FUNCTION_BLOCK FB_VISU_STOP_GATE
VAR_INPUT
END_VAR
VAR_OUTPUT
END_VAR
VAR
	iMoveCarrier: 		INT;
	bStopGateOpen: 		BOOL;
	bCarrierByStopGate: BOOL;
END_VAR

END_FUNCTION_BLOCK

(* stored: Version 1.1.0.1, ProductVersion 3.1.4024.12
   POU FB_VISU_STOP_GATE: Id {d2750194-f34b-4909-9964-9c58926728b0}, SpecialFunc None *)
